TYPE ST_Identity_PK1_OUT1 :
STRUCT
	ID	:STRING;
	ReadQuality:STRING;
END_STRUCT
END_TYPE

(* stored: Version 1.1.0.1, ProductVersion 3.1.4024.13
   DUT ST_Identity_PK1_OUT1: Id {aa868080-3c53-4b0c-91c2-a9fa64330134} *)
